TYPE ST_SAFETY_FBStatus :
STRUCT
	BUnknown						: BYTE;
	BState							: BYTE;
	wDiagnosis						: WORD;
	wInputs							: WORD; (* 1B - Restart, EDM... 2B - Safe inputs *)
	wOutputs						: WORD; (* 1B - Error, EDM... 2B - Safe inputs  *)
END_STRUCT
END_TYPE

(* stored: Version 1.1.0.1, ProductVersion 3.1.4022.12
   DUT ST_SAFETY_FBStatus: Id {cc89e3db-d6f3-4043-a4fe-50e8d6e43e4c} *)
